modbusMaster.Quantity := addresses[i].length;
modbusMaster.MBAddr := addresses[i].start;
modbusMaster.pMemoryAddr := ADR(values[offset]);
modbusMaster.Execute := execute;
CASE addresses[i].accessFunction OF
ReadCoils:
	length := (addresses[i].length + 7) / 8;
	modbusMaster.ReadCoils(cbLength := length);
ReadInputStatus:
	length := (addresses[i].length + 7) / 8;
	modbusMaster.ReadInputStatus(cbLength := length);
ReadInputRegs:
	length := 2 * addresses[i].length;
	modbusMaster.ReadInputRegs(cbLength := length);
END_CASE
modbusMasterBusy := modbusMaster.BUSY;
modbusMasterError := modbusMaster.Error;
modbusMasterErrorId := modbusMaster.ErrorId;
modbusMasterBytesRead := modbusMaster.cbRead;

IF modbusMasterBusy THEN
	execute := FALSE;
END_IF
modbusMasterReadyTrigger(CLK := modbusMasterBusy);

IF initScan THEN
	initScan := FALSE;
ELSE
	IF modbusMasterReadyTrigger.Q THEN
		offset := offset + length;
		i := i + 1;
		IF i >= n THEN
			initScan := TRUE;
			setValues := TRUE;
		ELSE
			execute := TRUE;
		END_IF
	END_IF
END_IF

IF setValues THEN
	j := 0;
	Heizkreis1_PumpeEin := values[j].0;
	Heizkreis2_PumpeEin := values[j].1;
	Heizkreis1_MischerAuf := values[j].2;
	Heizkreis1_MischerZu := values[j].3;
	Heizkreis2_MischerAuf := values[j].4;
	Heizkreis2_MischerZu := values[j].5;
	j := j + 1;
	Heizkreis0_PumpeEin := values[j].0;
	j := j + 1;
	Stoerung := values[j].4;
	j := j + 1;
	Heizkreis3_PumpeEin := values[j].1;
	Heizkreis4_PumpeEin := values[j].2;
	Heizkreis3_MischerAuf := values[j].3;
	Heizkreis3_MischerZu := values[j].4;
	Heizkreis4_MischerAuf := values[j].5;
	Heizkreis4_MischerZu := values[j].6;
	j := j + 1;
	TuerOffen := values[j].0;
	STB := values[j].1;
	NotAus := values[j].2;
	j := j + 1; KesselTemperatur := INT_TO_REAL(values[j]) / 2;
	j := j + 1; AbgasTemperatur := INT_TO_REAL(values[j]);
	j := j + 1; BoardTemperatur := INT_TO_REAL(values[j]) / 2;
	j := j + 1; RestSauerstoff := INT_TO_REAL(values[j]) / 10;
	j := j + 1; AussenTemperatur := INT_TO_REAL(values[j]) / 2;
	j := j + 3; SaugzugDrehzahl := INT_TO_REAL(values[j]);
	j := j + 1; StbTemperatur := INT_TO_REAL(values[j]) / 2;
	j := j + 1; Fuehler2Temperatur := INT_TO_REAL(values[j]) / 2;
	j := j + 6; Saugzug := INT_TO_REAL(values[j]);
	j := j + 3; Kesselstellgroesse := INT_TO_REAL(values[j]);
	j := j + 3; Heizkreis1_VoraufIst := INT_TO_REAL(values[j]) / 2;
	j := j + 1; Heizkreis1_VoraufSoll := INT_TO_REAL(values[j]) / 2;
	j := j + 1; Heizkreis1_Party := values[j];
	j := j + 1; Heizkreis1_RaumTemperatur := INT_TO_REAL(values[j]) / 2;
	j := j + 1; Heizkreis2_VoraufIst := INT_TO_REAL(values[j]) / 2;
	j := j + 1; Heizkreis2_VoraufSoll := INT_TO_REAL(values[j]) / 2;
	j := j + 1; Heizkreis2_Party := values[j];
	j := j + 1; Heizkreis2_RaumTemperatur := INT_TO_REAL(values[j]) / 2;
	j := j + 1; Heizkreis3_VoraufIst := INT_TO_REAL(values[j]) / 2;
	j := j + 1; Heizkreis3_VoraufSoll := INT_TO_REAL(values[j]) / 2;
	j := j + 1; Heizkreis3_Party := values[j];
	j := j + 1; Heizkreis3_RaumTemperatur := INT_TO_REAL(values[j]) / 2;
	j := j + 1; Heizkreis4_VoraufIst := INT_TO_REAL(values[j]) / 2;
	j := j + 1; Heizkreis4_VoraufSoll := INT_TO_REAL(values[j]) / 2;
	j := j + 1; Heizkreis4_Party := values[j];
	j := j + 1; Heizkreis4_RaumTemperatur := INT_TO_REAL(values[j]) / 2;
	j := j + 1; Boiler1_TemperaturOben := INT_TO_REAL(values[j]) / 2;
	j := j + 1; Boiler1_TemperaturSolarreferenz := INT_TO_REAL(values[j]) / 2;
	j := j + 1; Board_TemperaturPelletmodul := INT_TO_REAL(values[j]) / 2;
	j := j + 1; Betriebsstunden := values[j];
	setValues := FALSE;
END_IF
END_FUNCTION_BLOCK

(* POU FBs/FB_ANALYSE_VOLTAGE, ST *)
FUNCTION_BLOCK FB_ANALYSE_VOLTAGE
VAR_INPUT
	uliStartTimeNextLatch: ARRAY [0..1] OF UDINT;
	bWcState: BOOL;
END_VAR
VAR_IN_OUT
	iVoltage : ARRAY [0..9] OF INT;
END_VAR
VAR
	iBufferV: ARRAY [0..209] OF INT;
	iBufferT: ARRAY [0..209] OF T_DCTIME;
	i: INT;
	dctActSample: T_DCTIME;
	multiplier: T_DCTIME;
	dctSampleDelay: T_DCTIME;
	fbGETCURTASKINDEX: GETCURTASKINDEX;
	tCylceTime: T_DCTIME;
	tSampleTime: T_DCTIME;
	dctElSampleDelta: T_DCTIME;
	n: INT;
	m: INT;
	dctZeroPoint: ARRAY [1..2] OF T_DCTIME;
	bZeroPoint: ARRAY [1..2] OF BOOL;
	ui64Sub: T_ULARGE_INTEGER;
	ui64a: T_ULARGE_INTEGER;
	ui64b: T_ULARGE_INTEGER;
	dctZeroPointDelta: T_DCTIME;
	dctNextSample: T_DCTIME;
	uliStartTimeNextLatchLastCycle: ARRAY [0..1] OF UDINT;
	iBufferZeroSumV: INT;
	dctSampleTimePerV: T_DCTIME;
	dctSampleTimeOffset: T_DCTIME;
	ui64Add: T_ULARGE_INTEGER;
	diResultAdd: DINT;
	diResultSub: DINT;
	ui64Add1: T_ULARGE_INTEGER;
	ui64Sub1: T_ULARGE_INTEGER;
	ui64Cmp1: T_ULARGE_INTEGER;
	iActVoltage: INT;
	tHalfCylceTime: T_DCTIME;
	multi: T_ULARGE_INTEGER;
END_VAR
VAR_OUTPUT
	lrFrequency: LREAL;
	tNextZeroVoltage: T_DCTIME;
	bError: BOOL;
	bZeroFound: BOOL;
	bZeroNow: BOOL;
END_VAR
VAR CONSTANT
	uiOversampling: UINT := 10;
END_VAR
MEMCPY(ADR(dctNextSample), ADR(uliStartTimeNextLatch), SIZEOF(dctActsample));
MEMCPY(ADR(ui64a), ADR(dctNextSample), SIZEOF(ui64a));
MEMCPY(ADR(ui64b), ADR(dctActSample), SIZEOF(ui64b));
ui64Sub := UInt64Sub64(ui64a, ui64b);
MEMCPY(ADR(dctElSampleDelta), ADR(ui64Sub), SIZEOF(dctElSampleDelta));

fbGETCURTASKINDEX(index => );
tCylceTime.dwLowPart := SYSTEMTASKINFOARR[fbGETCURTASKINDEX.index].cycleTime * 100;
tCylceTime.dwHighPart := 0;


IF (dctElSampleDelta.dwLowPart <> tCylceTime.dwLowPart)
OR (dctElSampleDelta.dwHighPart <> tCylceTime.dwHighPart) THEN
	bError := TRUE;
ELSE
	bError := FALSE;
END_IF

IF NOT bWcState AND NOT bError THEN
	(* Samplezeit *)
	IF uiOversampling > 0 THEN
		tSampleTime.dwLowPart := (SYSTEMTASKINFOARR[fbGETCURTASKINDEX.index].cycleTime*100)/uiOversampling;
		tSampleTime.dwHighPart := 0;
	END_IF

	(* Spannungsspeicher befüllen *)
	FOR i := 10 TO 209 DO
		iBufferV[i-10] := iBufferV[i];
		iBufferT[i-10] := iBufferT[i];
	END_FOR

	FOR i := 200 TO 209 DO
		multiplier := LREAL_TO_UINT64(INT_TO_LREAL(i-200));
		dctSampleDelay := UInt64Mul64(tSampleTime, multiplier);
		iBufferT[i] := UInt64Add64(dctActSample, dctSampleDelay);
		iBufferV[i] := iVoltage[i-200];
	END_FOR

	(* Zeit der Nulldurchgänge bestimmen *)
	m := 208;
	bZeroPoint[1] := FALSE;
	bZeroPoint[2] := FALSE;
	bZeroNow := FALSE;
	iActVoltage := iBufferV[200];
	FOR n := 1 TO 2 DO
		FOR i := m TO 0 BY -1 DO
			IF (iBufferV[i].15 AND NOT iBufferV[i+1].15) OR (NOT iBufferV[i].15 AND iBufferV[i+1].15) THEN
				iBufferZeroSumV := ABS(iBufferV[i]) + ABS(iBufferV[i+1]);
				IF iBufferZeroSumV > 0 THEN
					dctSampleTimePerV.dwLowPart := LREAL_TO_DWORD(DWORD_TO_LREAL(tSampleTime.dwLowPart) / INT_TO_LREAL(iBufferZeroSumV));
					dctSampleTimePerV.dwHighPart := 0;
					dctSampleTimeOffset := UInt64Mul64(dctSampleTimePerV, LREAL_TO_UINT64(INT_TO_LREAL(ABS(iBufferV[i]))));
					dctZeroPoint[n] := UInt64Add64(iBufferT[i], dctSampleTimeOffset);
				ELSE
					dctZeroPoint[n] := iBufferT[i];
				END_IF

				m := i-1;

				bZeroPoint[n] := TRUE;
				IF n = 1 THEN
					multi.dwLowPart := 1;
					tHalfCylceTime.dwLowPart := tCylceTime.dwLowPart/2;
					ui64Add1 := UInt64Add64(UInt64Add64(dctZeroPoint[n],UInt64Mul64(dctZeroPointDelta, multi)), tHalfCylceTime);
					ui64Sub1 := UInt64Sub64(UInt64Add64(dctZeroPoint[n],UInt64Mul64(dctZeroPointDelta, multi)), tHalfCylceTime);
					ui64Cmp1 := F_GetActualDcTime();
					diResultAdd := UInt64Cmp64(ui64Cmp1, ui64Add1);
					diResultSub := UInt64Cmp64(ui64Cmp1, ui64Sub1);
					IF (diResultSub >= 0) AND (diResultAdd <= 0)THEN
						bZeroNow := TRUE;
					END_IF
				END_IF
				EXIT;
			END_IF
		END_FOR
	END_FOR
	IF bZeroPoint[1] AND bZeroPoint[2] THEN

		(* Berechnung des nächsten Nullpunkts *)
		MEMCPY(ADR(ui64a), ADR(dctZeroPoint[1]), SIZEOF(ui64a));
		MEMCPY(ADR(ui64b), ADR(dctZeroPoint[2]), SIZEOF(ui64b));
		ui64Sub := UInt64Sub64(ui64a, ui64b);
		MEMCPY(ADR(dctZeroPointDelta), ADR(ui64Sub), SIZEOF(dctZeroPointDelta));

		MEMCPY(ADR(ui64a), ADR(dctZeroPointDelta), SIZEOF(ui64a));
		MEMCPY(ADR(ui64b), ADR(dctZeroPoint), SIZEOF(ui64b));
		ui64Add := UInt64Add64(ui64a, ui64b);
		MEMCPY(ADR(tNextZeroVoltage), ADR(ui64Add), SIZEOF(tNextZeroVoltage));


		lrFrequency := 1 / (2 * DWORD_TO_LREAL(dctZeroPointDelta.dwLowPart) / 1000000000);
	END_IF
END_IF
MEMCPY(ADR(dctActSample), ADR(uliStartTimeNextLatch), SIZEOF(dctActsample));

uliStartTimeNextLatchLastCycle := uliStartTimeNextLatch;
END_FUNCTION_BLOCK

(* POU FBs/FB_SYNC_RELAIS, ST *)
FUNCTION_BLOCK FB_SYNC_RELAIS
VAR_INPUT
	bValue: BOOL;
	udiDelayNanoSek: UDINT;
	tNextZeroVoltage: T_DCTIME;
END_VAR
VAR_OUTPUT
	bRelay AT %Q*: BOOL;
END_VAR
VAR
	fbGETCURTASKINDEX: GETCURTASKINDEX;
	tNextZeroVoltageLast: T_DCTIME;
	TON_FAILURE: TON;
	TOF_WAIT: TOF;
	udiLastOnlineChangeCount: UDINT;
	multi: T_DCTIME;
	ui64Add1: T_ULARGE_INTEGER;
	tHalfCylceTime: T_DCTIME;
	ui64Sub1: T_ULARGE_INTEGER;
	ui64Cmp1: T_ULARGE_INTEGER;
	diResultAdd: DINT;
	diResultSub: DINT;
	tCylceTime: T_DCTIME;
END_VAR
(*fTvalue(CLK:=bValue AND bRelay);
IF fTvalue.Q OR bReset THEN
	bRelay := FALSE;
	bReset := FALSE;
END_IF
*)

TON_FAILURE(IN := tNextZeroVoltage.dwLowPart = tNextZeroVoltageLast.dwLowPart, PT := t#100ms);
tNextZeroVoltageLast.dwLowPart := tNextZeroVoltage.dwLowPart;

TOF_WAIT(IN := SYSTEMINFO.onlineChangeCount <> udiLastOnlineChangeCount, PT := t#0.5s);
udiLastOnlineChangeCount := SYSTEMINFO.onlineChangeCount;

IF bValue AND NOT bRelay AND NOT TON_FAILURE.Q THEN
	fbGETCURTASKINDEX(index => );
	tCylceTime.dwLowPart := SYSTEMTASKINFOARR[fbGETCURTASKINDEX.index].cycleTime * 100;
	tCylceTime.dwHighPart := 0;

	multi.dwLowPart := udiDelayNanoSek;
	tHalfCylceTime.dwLowPart := tCylceTime.dwLowPart/2;
	ui64Add1 := UInt64Add64(UInt64Sub64(tNextZeroVoltage, multi), tHalfCylceTime);
	ui64Sub1 := UInt64Sub64(UInt64Sub64(tNextZeroVoltage, multi), tHalfCylceTime);
	ui64Cmp1 := F_GetActualDcTime();
	diResultAdd := UInt64Cmp64(ui64Cmp1, ui64Add1);
	diResultSub := UInt64Cmp64(ui64Cmp1, ui64Sub1);

	IF (diResultSub >= 0) AND (diResultAdd <= 0) THEN
		bRelay := TRUE;
	END_IF
END_IF

IF NOT bValue AND bRelay AND NOT TON_FAILURE.Q THEN
	fbGETCURTASKINDEX(index => );
	tCylceTime.dwLowPart := SYSTEMTASKINFOARR[fbGETCURTASKINDEX.index].cycleTime * 100;
	tCylceTime.dwHighPart := 0;

	multi.dwLowPart := udiDelayNanoSek / 2;
	tHalfCylceTime.dwLowPart := tCylceTime.dwLowPart / 2;
	ui64Add1 := UInt64Add64(UInt64Sub64(tNextZeroVoltage, multi), tHalfCylceTime);
	ui64Sub1 := UInt64Sub64(UInt64Sub64(tNextZeroVoltage, multi), tHalfCylceTime);
	ui64Cmp1 := F_GetActualDcTime();
	diResultAdd := UInt64Cmp64(ui64Cmp1, ui64Add1);
	diResultSub := UInt64Cmp64(ui64Cmp1, ui64Sub1);

	IF (diResultSub >= 0) AND (diResultAdd <= 0)THEN
		bRelay := FALSE;
	END_IF
END_IF
END_FUNCTION_BLOCK

(* POU FBs/FB_Modbus_RTU_Master_KL6x22B, ST *)
FUNCTION_BLOCK FB_Modbus_RTU_Master_KL6x22B
VAR_INPUT
	bStart: BOOL; (* Start Modbus-Communication *)
	byModbusSlaveStartAdress: BYTE := 1; (* First Modbus Device Address *)
	byModbusSlaveEndAdress: BYTE := 247; (* Last Modbus Device Address *)
	tModbusSlaveTimeout: TIME := t#500ms; (* Modbus Communication Timeout *)
	tDelayModbusTime: TIME := t#50ms; (* Delay between two Modbus Requests *)
	bIgnoreError: BOOL; (* Ignore ever Modbus Error *)
END_VAR
VAR_OUTPUT
	bBusy: BOOL; (* if TRUE, Modbustelegramms are being sent *)
	bError: BOOL; (* if TRUE, a Modbustelegramm wasn't send correctly *)
	eErrorID: MODBUS_ERRORS;
	bNoResponse: BOOL; (* if TRUE, a FB with a DeviceAddress isn't existing as phyical device *)
	byLastNoResponseModbusAddress: BYTE;
END_VAR
VAR_IN_OUT
	stCommunication: stFB_ModbusMaster; (* Communicationvariable must connect with ever Slave FB *)
END_VAR
VAR
	FB_ModbusRtuMaster_KL6x22B: ModbusRtuMaster_KL6x22B;
	R_TRIG_START: R_TRIG;
	F_TRIG_ModbusReady: F_TRIG;
	TON_Delay: TON;
	i: INT;
	j: INT;
	bBusyMaster: BOOL;
	bNextModbusDevice: BOOL;
	bNextData: BOOL;
END_VAR
R_TRIG_START(CLK := bStart);
TON_Delay(IN := i = 2, PT := tDelayModbusTime);

F_TRIG_ModbusReady(CLK := FB_ModbusRtuMaster_KL6x22B.BUSY);
IF F_TRIG_ModbusReady.Q THEN
	bBusy := FALSE;
END_IF

(* Init FB *)
IF R_TRIG_START.Q THEN
	i := 0;
END_IF

CASE i OF
0: (* Set Startaddress *)
	IF R_TRIG_START.Q THEN
		bBusy := TRUE;
		bError := FALSE;
		eErrorID := 0;
		stCommunication.byCurrentModbusSlaveAdress := byModbusSlaveStartAdress;
		i := i + 1;
	END_IF
1: (* Exist Address?*)
	IF stCommunication.bModbusAddressExist THEN
		i := i + 1;
		stCommunication.bModbusCommunicationActive := TRUE;
	ELSE
		j := j + 1;
	END_IF
	IF j > 10 THEN
		stCommunication.byCurrentModbusSlaveAdress := stCommunication.byCurrentModbusSlaveAdress + 1;
		j := 0;
	END_IF
	IF stCommunication.byCurrentModbusSlaveAdress > byModbusSlaveEndAdress OR stCommunication.byCurrentModbusSlaveAdress > 247 THEN
		stCommunication.byCurrentModbusSlaveAdress := byModbusSlaveStartAdress;
		IF byModbusSlaveStartAdress < 1 THEN
			stCommunication.byCurrentModbusSlaveAdress := 1;
		END_IF
	END_IF

2: (* Init Modbus and order data from slave*)
	IF TON_Delay.Q AND bStart THEN
		bBusy := TRUE;
		bError := FALSE;
		eErrorID := 0;
		FB_ModbusRtuMaster_KL6x22B.ReadCoils(Execute := FALSE);
		FB_ModbusRtuMaster_KL6x22B.ReadInputStatus(Execute := FALSE);
		FB_ModbusRtuMaster_KL6x22B.ReadRegs(Execute := FALSE);
		FB_ModbusRtuMaster_KL6x22B.ReadInputRegs(Execute := FALSE);
		FB_ModbusRtuMaster_KL6x22B.WriteSingleCoil(Execute := FALSE);
		FB_ModbusRtuMaster_KL6x22B.WriteSingleRegister(Execute := FALSE);
		FB_ModbusRtuMaster_KL6x22B.Diagnostics(Execute := FALSE);
		FB_ModbusRtuMaster_KL6x22B.WriteMultipleCoils(Execute := FALSE);
		FB_ModbusRtuMaster_KL6x22B.WriteRegs(Execute := FALSE);
		i := i + 1;
	END_IF
3: (*Wait for new data from slave *)
	CASE stCommunication.stCurrentDeviceSpace[0].iModbusFunction OF
		1:
			FB_ModbusRtuMaster_KL6x22B.ReadCoils(
				UnitID:=stCommunication.byCurrentModbusSlaveAdress,
				Quantity:= stCommunication.stCurrentDeviceSpace[0].wSPSDataSpaceLength/2,
				MBAddr:= stCommunication.stCurrentDeviceSpace[0].wModbusAdress,
				cbLength:= stCommunication.stCurrentDeviceSpace[0].wSPSDataSpaceLength,
				pMemoryAddr:= stCommunication.stCurrentDeviceSpace[0].pSPSDataSpace,
				Execute:= TRUE,
				Timeout := tModbusSlaveTimeout,
				Busy=>bBusyMaster);
		2:
			FB_ModbusRtuMaster_KL6x22B.ReadInputStatus(
				UnitID:=stCommunication.byCurrentModbusSlaveAdress,
				Quantity:= stCommunication.stCurrentDeviceSpace[0].wSPSDataSpaceLength/2,
				MBAddr:= stCommunication.stCurrentDeviceSpace[0].wModbusAdress,
				cbLength:= stCommunication.stCurrentDeviceSpace[0].wSPSDataSpaceLength,
				pMemoryAddr:= stCommunication.stCurrentDeviceSpace[0].pSPSDataSpace,
				Execute:= TRUE,
				Timeout := tModbusSlaveTimeout,
				Busy=>bBusyMaster);
		3:
			FB_ModbusRtuMaster_KL6x22B.ReadRegs(
				UnitID:=stCommunication.byCurrentModbusSlaveAdress,
				Quantity:= stCommunication.stCurrentDeviceSpace[0].wSPSDataSpaceLength/2,
				MBAddr:= stCommunication.stCurrentDeviceSpace[0].wModbusAdress,
				cbLength:= stCommunication.stCurrentDeviceSpace[0].wSPSDataSpaceLength,
				pMemoryAddr:= stCommunication.stCurrentDeviceSpace[0].pSPSDataSpace,
				Execute:= TRUE,
				Timeout := tModbusSlaveTimeout,
				Busy=>bBusyMaster);
		4:
			FB_ModbusRtuMaster_KL6x22B.ReadInputRegs(
				UnitID:=stCommunication.byCurrentModbusSlaveAdress,
				Quantity:= stCommunication.stCurrentDeviceSpace[0].wSPSDataSpaceLength/2,
				MBAddr:= stCommunication.stCurrentDeviceSpace[0].wModbusAdress,
				cbLength:= stCommunication.stCurrentDeviceSpace[0].wSPSDataSpaceLength,
				pMemoryAddr:= stCommunication.stCurrentDeviceSpace[0].pSPSDataSpace,
				Execute:= TRUE,
				Timeout := tModbusSlaveTimeout,
				Busy=>bBusyMaster);
		5:
			FB_ModbusRtuMaster_KL6x22B.WriteSingleCoil(
				UnitID:=stCommunication.byCurrentModbusSlaveAdress,
				Quantity:= stCommunication.stCurrentDeviceSpace[0].wSPSDataSpaceLength/2,
				MBAddr:= stCommunication.stCurrentDeviceSpace[0].wModbusAdress,
				cbLength:= stCommunication.stCurrentDeviceSpace[0].wSPSDataSpaceLength,
				pMemoryAddr:= stCommunication.stCurrentDeviceSpace[0].pSPSDataSpace,
				Execute:= TRUE,
				Timeout := tModbusSlaveTimeout,
				Busy=>bBusyMaster);
		6:
			FB_ModbusRtuMaster_KL6x22B.WriteSingleRegister(
				UnitID:=stCommunication.byCurrentModbusSlaveAdress,
				Quantity:= stCommunication.stCurrentDeviceSpace[0].wSPSDataSpaceLength/2,
				MBAddr:= stCommunication.stCurrentDeviceSpace[0].wModbusAdress,
				cbLength:= stCommunication.stCurrentDeviceSpace[0].wSPSDataSpaceLength,
				pMemoryAddr:= stCommunication.stCurrentDeviceSpace[0].pSPSDataSpace,
				Execute:= TRUE,
				Timeout := tModbusSlaveTimeout,
				Busy=>bBusyMaster);
		8:
			FB_ModbusRtuMaster_KL6x22B.Diagnostics(
				UnitID:=stCommunication.byCurrentModbusSlaveAdress,
				Quantity:= stCommunication.stCurrentDeviceSpace[0].wSPSDataSpaceLength/2,
				MBAddr:= stCommunication.stCurrentDeviceSpace[0].wModbusAdress,
				cbLength:= stCommunication.stCurrentDeviceSpace[0].wSPSDataSpaceLength,
				pMemoryAddr:= stCommunication.stCurrentDeviceSpace[0].pSPSDataSpace,
				Execute:= TRUE,
				Timeout := tModbusSlaveTimeout,
				Busy=>bBusyMaster);
		15:
			FB_ModbusRtuMaster_KL6x22B.WriteMultipleCoils(
				UnitID:=stCommunication.byCurrentModbusSlaveAdress,
				Quantity:= stCommunication.stCurrentDeviceSpace[0].wSPSDataSpaceLength/2,
				MBAddr:= stCommunication.stCurrentDeviceSpace[0].wModbusAdress,
				cbLength:= stCommunication.stCurrentDeviceSpace[0].wSPSDataSpaceLength,
				pMemoryAddr:= stCommunication.stCurrentDeviceSpace[0].pSPSDataSpace,
				Execute:= TRUE,
				Timeout := tModbusSlaveTimeout,
				Busy=>bBusyMaster);
		16:
			FB_ModbusRtuMaster_KL6x22B.WriteRegs(
				UnitID:=stCommunication.byCurrentModbusSlaveAdress,
				Quantity:= stCommunication.stCurrentDeviceSpace[0].wSPSDataSpaceLength/2,
				MBAddr:= stCommunication.stCurrentDeviceSpace[0].wModbusAdress,
				cbLength:= stCommunication.stCurrentDeviceSpace[0].wSPSDataSpaceLength,
				pMemoryAddr:= stCommunication.stCurrentDeviceSpace[0].pSPSDataSpace,
				Execute:= TRUE,
				Timeout := tModbusSlaveTimeout,
				Busy=>bBusyMaster);
	ELSE
		bError := TRUE;
		eErrorID := 1;
	END_CASE

	IF F_TRIG_ModbusReady.Q AND NOT FB_ModbusRtuMaster_KL6x22B.Error THEN (*No Error*)
		bNoResponse := FALSE;
		bError := FALSE;
		bNextData := TRUE;
	ELSIF FB_ModbusRtuMaster_KL6x22B.Error AND FB_ModbusRtuMaster_KL6x22B.ErrorId = 16#25 THEN (*no  Response *)
		i := 1;
		bNoResponse := TRUE;
		bError := TRUE;
		eErrorID := FB_ModbusRtuMaster_KL6x22B.ErrorId;
		byLastNoResponseModbusAddress := stCommunication.byCurrentModbusSlaveAdress;
		stCommunication.byCurrentModbusSlaveAdress := stCommunication.byCurrentModbusSlaveAdress + 1;
		stCommunication.bModbusAddressExist := FALSE;
		stCommunication.bModbusCommunicationActive := FALSE;
		i := 1;
		FOR j := 0 TO stCommunication.iNumberOfData DO
			stCommunication.stCurrentDeviceSpace[stCommunication.iNumberOfData].iModbusFunction := 0;
			stCommunication.stCurrentDeviceSpace[stCommunication.iNumberOfData].pSPSDataSpace := 0;
			stCommunication.stCurrentDeviceSpace[stCommunication.iNumberOfData].wModbusAdress := 0;
			stCommunication.stCurrentDeviceSpace[stCommunication.iNumberOfData].wSPSDataSpaceLength := 0;
		END_FOR
	ELSIF FB_ModbusRtuMaster_KL6x22B.Error AND bIgnoreError THEN
		bNoResponse := FALSE;
		bError := TRUE;
		bNextData := TRUE;
	ELSIF FB_ModbusRtuMaster_KL6x22B.Error THEN
		i := 100;
	END_IF

	IF bNextData THEN
		FOR j := 1 TO stCommunication.iNumberOfData DO
			stCommunication.stCurrentDeviceSpace[j-1] := stCommunication.stCurrentDeviceSpace[j];
		END_FOR
		stCommunication.stCurrentDeviceSpace[stCommunication.iNumberOfData].iModbusFunction := 0;
		stCommunication.stCurrentDeviceSpace[stCommunication.iNumberOfData].pSPSDataSpace := 0;
		stCommunication.stCurrentDeviceSpace[stCommunication.iNumberOfData].wModbusAdress := 0;
		stCommunication.stCurrentDeviceSpace[stCommunication.iNumberOfData].wSPSDataSpaceLength := 0;
		i := 2;
		bNextData := FALSE;
		bBusy := FALSE;
		IF stCommunication.stCurrentDeviceSpace[0].iModbusFunction = 0 THEN
			stCommunication.byCurrentModbusSlaveAdress := stCommunication.byCurrentModbusSlaveAdress + 1;
			stCommunication.bModbusAddressExist := FALSE;
			stCommunication.bModbusCommunicationActive := FALSE;
			i := 1;
		END_IF
	END_IF
100:
	bError := FB_ModbusRtuMaster_KL6x22B.Error;
	eErrorID := FB_ModbusRtuMaster_KL6x22B.ErrorId;
END_CASE
END_FUNCTION_BLOCK

(* POU FBs/FB_ScanModbusSlaveAdresses_KL6x22B, ST *)
FUNCTION_BLOCK FB_ScanModbusSlaveAdresses_KL6x22B
VAR_INPUT
	bStartScan: BOOL; (* Start scanning *)
	bOnlyRead: BOOL;
	byModbusSlaveDeviceAdress: BYTE := 1; (* Modbus Device Address *)
	MBStartAddr: WORD := 0; (* First ModbusRegisterAddress *)
	MBEndAddr: WORD := 100; (* Last ModbusRegisterAddress *)
	(* ATTENTION please!!! This FB writes to the ModbusRegisterAddress
		the value 0 with every write function!!!
		DON'T SCAN SYSTEMREGISTER OR FIRMWARE REGISTER
		... the Device could be destroyed! *)
END_VAR
VAR_OUTPUT
	rPercentOfScanProzess: REAL;
	bNoFreeSpaceForNewValues: BOOL;
	bReady: BOOL;
	stValues: ARRAY [0..999] OF stResultOfModbusSlaveScan; (* Scanresult *)
END_VAR
VAR
	FB_ModbusRtuMaster_KL6x22B: ModbusRtuMaster_KL6x22B;
	F_TRIG1: F_TRIG;
	R_TRIG1: R_TRIG;
	F_TRIG2: F_TRIG;
	bStart: BOOL;
	MBFunction: INT := 1;
	MBAddr: WORD;
	Pos: INT;
	i: INT;
	Result: UDINT;
	rActuellScanProzess: REAL;
END_VAR
CASE MBFunction OF
1:
	FB_ModbusRtuMaster_KL6x22B.ReadCoils(
		UnitID := byModbusSlaveDeviceAdress,
		Quantity := 1,
		MBAddr := MBAddr,
		cbLength := 2,
		pMemoryAddr := ADR(stValues[Pos].wValue),
		Execute := bStart,
		Timeout := t#1s,
		BUSY => ,
		Error => ,
		ErrorId => ,
		cbRead => );
2:
	FB_ModbusRtuMaster_KL6x22B.ReadInputStatus(
		UnitID:=byModbusSlaveDeviceAdress ,
		Quantity:=1 ,
		MBAddr:=MBAddr ,
		cbLength:=2 ,
		pMemoryAddr:=ADR(stValues[Pos].wValue) ,
		Execute:=bStart ,
		Timeout:=t#1s ,
		BUSY=> ,
		Error=> ,
		ErrorId=> ,
		cbRead=> );
3:
	FB_ModbusRtuMaster_KL6x22B.ReadRegs(
		UnitID:=byModbusSlaveDeviceAdress ,
		Quantity:=1 ,
		MBAddr:=MBAddr ,
		cbLength:=2 ,
		pMemoryAddr:=ADR(stValues[Pos].wValue) ,
		Execute:=bStart ,
		Timeout:=t#1s ,
		BUSY=> ,
		Error=> ,
		ErrorId=> ,
		cbRead=> );
4:
	FB_ModbusRtuMaster_KL6x22B.ReadInputRegs(
		UnitID:=byModbusSlaveDeviceAdress ,
		Quantity:=1 ,
		MBAddr:=MBAddr ,
		cbLength:=2 ,
		pMemoryAddr:=ADR(stValues[Pos].wValue) ,
		Execute:=bStart ,
		Timeout:=t#1s ,
		BUSY=> ,
		Error=> ,
		ErrorId=> ,
		cbRead=> );
5:
	FB_ModbusRtuMaster_KL6x22B.WriteSingleCoil(
		UnitID:=byModbusSlaveDeviceAdress ,
		Quantity:=1 ,
		MBAddr:=MBAddr ,
		cbLength:=2 ,
		pMemoryAddr:=ADR(stValues[Pos].wValue) ,
		Execute:=bStart ,
		Timeout:=t#1s ,
		BUSY=> ,
		Error=> ,
		ErrorId=> ,
		cbRead=> );
6:
	FB_ModbusRtuMaster_KL6x22B.WriteSingleRegister(
		UnitID:=byModbusSlaveDeviceAdress ,
		Quantity:=1 ,
		MBAddr:=MBAddr ,
		cbLength:=2 ,
		pMemoryAddr:=ADR(stValues[Pos].wValue) ,
		Execute:=bStart ,
		Timeout:=t#1s ,
		BUSY=> ,
		Error=> ,
		ErrorId=> ,
		cbRead=> );
8:
	FB_ModbusRtuMaster_KL6x22B.Diagnostics(
		UnitID:=byModbusSlaveDeviceAdress ,
		Quantity:=1 ,
		MBAddr:=MBAddr ,
		cbLength:=2 ,
		pMemoryAddr:=ADR(stValues[Pos].wValue) ,
		Execute:=bStart ,
		Timeout:=t#1s ,
		BUSY=> ,
		Error=> ,
		ErrorId=> ,
		cbRead=> );
15:
	FB_ModbusRtuMaster_KL6x22B.WriteMultipleCoils(
		UnitID:=byModbusSlaveDeviceAdress ,
		Quantity:=1 ,
		MBAddr:=MBAddr ,
		cbLength:=2 ,
		pMemoryAddr:=ADR(stValues[Pos].wValue) ,
		Execute:=bStart ,
		Timeout:=t#1s ,
		BUSY=> ,
		Error=> ,
		ErrorId=> ,
		cbRead=> );
16:
	FB_ModbusRtuMaster_KL6x22B.WriteRegs(
		UnitID:=byModbusSlaveDeviceAdress ,
		Quantity:=1 ,
		MBAddr:=MBAddr ,
		cbLength:=2 ,
		pMemoryAddr:=ADR(stValues[Pos].wValue) ,
		Execute:=bStart ,
		Timeout:=t#1s ,
		BUSY=> ,
		Error=> ,
		ErrorId=> ,
		cbRead=> );
END_CASE

F_TRIG1(CLK := FB_ModbusRtuMaster_KL6x22B.BUSY);

R_TRIG1(CLK := bStartScan);
F_TRIG2(CLK := bStartScan);

IF F_TRIG2.Q THEN
	i := 0;
END_IF

CASE i OF
0:
	IF R_TRIG1.Q THEN
		i := i + 1;
		bStart := FALSE;
		bNoFreeSpaceForNewValues := FALSE;
		bReady := FALSE;
		MBAddr := MBStartAddr;
		rPercentOfScanProzess := 0.0;
		rActuellScanProzess := 0.0;
	END_IF
1:
	bStart := TRUE;
	i := i + 1;
2:
	IF F_TRIG1.Q AND ((NOT FB_ModbusRtuMaster_KL6x22B.Error) OR FB_ModbusRtuMaster_KL6x22B.ErrorId = 3) THEN
		stValues[Pos].eModbusError := FB_ModbusRtuMaster_KL6x22B.ErrorId;
		stValues[Pos].eModbusfunction := MBFunction;
		stValues[Pos].iModbusAdress := MBAddr;
		(*New Array Position*)
		Pos := Pos + 1;
	END_IF

	IF F_TRIG1.Q THEN
		IF Pos > 999 THEN
			Pos := 0;
			i := 0;
			bNoFreeSpaceForNewValues := TRUE;
		END_IF

		MBAddr := MBAddr + 1;
		i := 1;
		bStart := FALSE;
		IF MBAddr > MBEndAddr THEN
			MBAddr := MBStartAddr;
			MBFunction := MBFunction + 1;
			IF MBFunction > 4 AND bOnlyRead OR MBFunction = 17 THEN
				MBFunction := 1;
				i := 4;
				bReady := TRUE;
			ELSE
				IF MBFunction = 7 THEN
					MBFunction := 8;
				ELSIF MBFunction = 9 THEN
					MBFunction := 15;
				ELSE
					;
				END_IF
			END_IF
		END_IF
	END_IF
4:
		rPercentOfScanProzess := 100.0;
END_CASE

IF F_TRIG1.Q THEN
	rActuellScanProzess := rActuellScanProzess + 1.0;
END_IF

IF NOT (i = 4) THEN
	rPercentOfScanProzess := (100.0 * rActuellScanProzess) / (9.0 * WORD_TO_REAL(MBEndAddr - MBStartAddr));
END_IF
END_FUNCTION_BLOCK

(* POU FBs/FB_Toggle, ST *)
FUNCTION_BLOCK FB_Toggle
VAR_INPUT
	onTime: TIME :=  t#0.5s;
	offTime: TIME := t#1s;
END_VAR
VAR_OUTPUT
	Q: BOOL;
END_VAR
VAR
	t1: TON;
	t2: TOF;
END_VAR
t1(IN := NOT t2.Q, pt := offTime);
t2(IN := t1.Q, pt := onTime);
Q := t2.Q;

(* c.henke variant:
TON1(IN := NOT TON1.Q AND bStart, PT := t#1s);
IF TON1.Q THEN
	bRelayPLC := NOT bRelayPLC;
END_IF
*)
END_FUNCTION_BLOCK

(* Visualisation VI_BACKGROUND
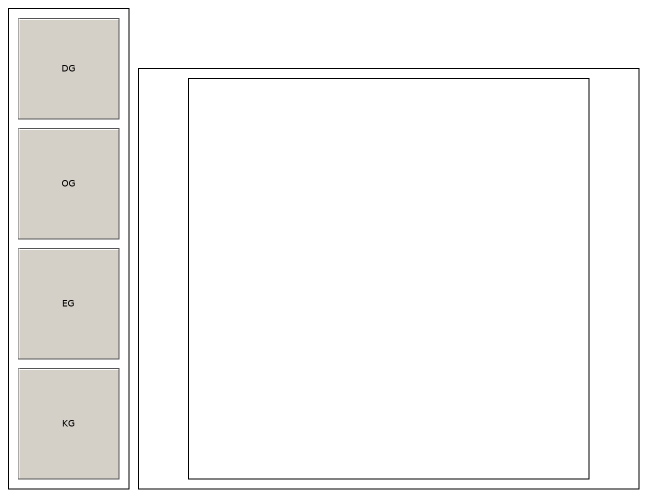
button at (10,360)-(111,471): text "KG"; opens vi_KG
button at (10,240)-(111,351): text "EG"; opens vi_EG
button at (10,120)-(111,231): text "OG"; opens vi_OG
button at (10,10)-(111,111): text "DG"; opens vi_DG
3 more shapes without text or variables
*)

(* Visualisation templates/VI_BUTTONDOUBLE
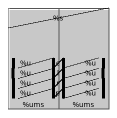
button at (50,0)-(101,101): text "%ums"; shows $fbButton_R$.LONGPRESS; taps $fbButton_R$.viIN
button at (0,0)-(51,101): text "%ums"; shows $fbButton_L$.LONGPRESS; taps $fbButton_L$.viIN
curve at (55,80)-(90,90): text "%u"; shows $fbButton_R$.usageCounterPress
curve at (95,80)-(95,90): alarm colour if $fbButton_R$.toggleOnPress
curve at (95,70)-(95,80): alarm colour if $fbButton_R$.toggleOnRelease
curve at (95,60)-(95,70): alarm colour if $fbButton_R$.toggleOnLongpress
curve at (95,50)-(95,60): alarm colour if $fbButton_R$.toggleOnClick
curve at (55,70)-(90,80): text "%u"; shows $fbButton_R$.usageCounterRelease
curve at (55,60)-(90,70): text "%u"; shows $fbButton_R$.usageCounterLongpress
curve at (55,50)-(90,60): text "%u"; shows $fbButton_R$.usageCounterClick
curve at (55,80)-(55,90): alarm colour if $fbButton_R$.isPressed
curve at (55,70)-(55,80): alarm colour if $fbButton_R$.isReleased
curve at (55,60)-(55,70): alarm colour if $fbButton_R$.isLongpressed
curve at (55,50)-(55,60): alarm colour if $fbButton_R$.isClicked
curve at (45,50)-(55,60): text "c"
curve at (45,60)-(55,70): text "l"
curve at (45,70)-(55,80): text "r"
curve at (45,80)-(55,90): text "p"
curve at (10,80)-(45,90): text "%u"; shows $fbButton_L$.usageCounterPress
curve at (5,80)-(5,90): alarm colour if $fbButton_L$.toggleOnPress
curve at (5,70)-(5,80): alarm colour if $fbButton_L$.toggleOnRelease
curve at (5,60)-(5,70): alarm colour if $fbButton_L$.toggleOnLongpress
curve at (5,50)-(5,60): alarm colour if $fbButton_L$.toggleOnClick
curve at (10,70)-(45,80): text "%u"; shows $fbButton_L$.usageCounterRelease
curve at (10,60)-(45,70): text "%u"; shows $fbButton_L$.usageCounterLongpress
curve at (10,50)-(45,60): text "%u"; shows $fbButton_L$.usageCounterClick
curve at (45,80)-(45,90): alarm colour if $fbButton_L$.isPressed
curve at (45,70)-(45,80): alarm colour if $fbButton_L$.isReleased
curve at (45,60)-(45,70): alarm colour if $fbButton_L$.isLongpressed
curve at (45,50)-(45,60): alarm colour if $fbButton_L$.isClicked
curve at (0,0)-(100,20): text "%s"; shows $fbButton_L$.viText
*)

(* Visualisation templates/vi_ButtonDouble_tiny
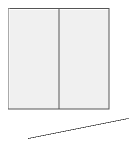
button at (50,0)-(101,101): taps $fbButton_R$.viIN
button at (0,0)-(51,101): taps $fbButton_L$.viIN
1 more shapes without text or variables
*)

(* Visualisation templates/vi_ButtonSingle
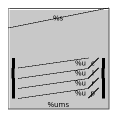
button at (0,0)-(101,101): text "%ums"; shows $fbButton$.LONGPRESS; taps $fbButton$.viIN
curve at (0,0)-(100,20): text "%s"; shows $fbButton$.viText
curve at (10,80)-(80,90): text "%u"; shows $fbButton$.usageCounterPress
curve at (95,80)-(95,90): alarm colour if $fbButton$.toggleOnPress
curve at (95,70)-(95,80): alarm colour if $fbButton$.toggleOnRelease
curve at (95,60)-(95,70): alarm colour if $fbButton$.toggleOnLongpress
curve at (95,50)-(95,60): alarm colour if $fbButton$.toggleOnClick
curve at (10,70)-(80,80): text "%u"; shows $fbButton$.usageCounterRelease
curve at (10,60)-(80,70): text "%u"; shows $fbButton$.usageCounterLongpress
curve at (10,50)-(80,60): text "%u"; shows $fbButton$.usageCounterClick
curve at (80,50)-(90,60): text "c"
curve at (80,60)-(90,70): text "l"
curve at (80,70)-(90,80): text "r"
curve at (80,80)-(90,90): text "p"
curve at (5,80)-(5,90): alarm colour if $fbButton$.isPressed
curve at (5,70)-(5,80): alarm colour if $fbButton$.isReleased
curve at (5,60)-(5,70): alarm colour if $fbButton$.isLongpressed
curve at (5,50)-(5,60): alarm colour if $fbButton$.isClicked
*)

(* Visualisation templates/vi_ButtonSingle_tiny
button at (0,0)-(101,101): taps $fbButton$.viIN
*)

(* Visualisation templates/vi_ButtonTripple
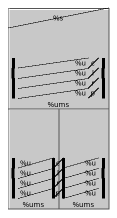
button at (50,100)-(101,201): text "%ums"; shows $fbButton_R$.LONGPRESS; taps $fbButton_R$.viIN
button at (0,100)-(51,201): text "%ums"; shows $fbButton_L$.LONGPRESS; taps $fbButton_L$.viIN
curve at (55,180)-(90,190): text "%u"; shows $fbButton_R$.usageCounterPress
curve at (95,180)-(95,190): alarm colour if $fbButton_R$.toggleOnPress
curve at (95,170)-(95,180): alarm colour if $fbButton_R$.toggleOnRelease
curve at (95,160)-(95,170): alarm colour if $fbButton_R$.toggleOnLongpress
curve at (95,150)-(95,160): alarm colour if $fbButton_R$.toggleOnClick
curve at (55,170)-(90,180): text "%u"; shows $fbButton_R$.usageCounterRelease
curve at (55,160)-(90,170): text "%u"; shows $fbButton_R$.usageCounterLongpress
curve at (55,150)-(90,160): text "%u"; shows $fbButton_R$.usageCounterClick
curve at (55,180)-(55,190): alarm colour if $fbButton_R$.isPressed
curve at (55,170)-(55,180): alarm colour if $fbButton_R$.isReleased
curve at (55,160)-(55,170): alarm colour if $fbButton_R$.isLongpressed
curve at (55,150)-(55,160): alarm colour if $fbButton_R$.isClicked
curve at (45,150)-(55,160): text "c"
curve at (45,160)-(55,170): text "l"
curve at (45,170)-(55,180): text "r"
curve at (45,180)-(55,190): text "p"
curve at (10,180)-(45,190): text "%u"; shows $fbButton_L$.usageCounterPress
curve at (5,180)-(5,190): alarm colour if $fbButton_L$.toggleOnPress
curve at (5,170)-(5,180): alarm colour if $fbButton_L$.toggleOnRelease
curve at (5,160)-(5,170): alarm colour if $fbButton_L$.toggleOnLongpress
curve at (5,150)-(5,160): alarm colour if $fbButton_L$.toggleOnClick
curve at (10,170)-(45,180): text "%u"; shows $fbButton_L$.usageCounterRelease
curve at (10,160)-(45,170): text "%u"; shows $fbButton_L$.usageCounterLongpress
curve at (10,150)-(45,160): text "%u"; shows $fbButton_L$.usageCounterClick
curve at (45,180)-(45,190): alarm colour if $fbButton_L$.isPressed
curve at (45,170)-(45,180): alarm colour if $fbButton_L$.isReleased
curve at (45,160)-(45,170): alarm colour if $fbButton_L$.isLongpressed
curve at (45,150)-(45,160): alarm colour if $fbButton_L$.isClicked
button at (0,0)-(101,101): text "%ums"; shows $fbButton_T$.LONGPRESS; taps $fbButton_T$.viIN
curve at (0,0)-(100,20): text "%s"; shows $fbButton_T$.viText
curve at (10,80)-(80,90): text "%u"; shows $fbButton_T$.usageCounterPress
curve at (95,80)-(95,90): alarm colour if $fbButton_T$.toggleOnPress
curve at (95,70)-(95,80): alarm colour if $fbButton_T$.toggleOnRelease
curve at (95,60)-(95,70): alarm colour if $fbButton_T$.toggleOnLongpress
curve at (95,50)-(95,60): alarm colour if $fbButton_T$.toggleOnClick
curve at (10,70)-(80,80): text "%u"; shows $fbButton_T$.usageCounterRelease
curve at (10,60)-(80,70): text "%u"; shows $fbButton_T$.usageCounterLongpress
curve at (10,50)-(80,60): text "%u"; shows $fbButton_T$.usageCounterClick
curve at (80,50)-(90,60): text "c"
curve at (80,60)-(90,70): text "l"
curve at (80,70)-(90,80): text "r"
curve at (80,80)-(90,90): text "p"
curve at (5,80)-(5,90): alarm colour if $fbButton_T$.isPressed
curve at (5,70)-(5,80): alarm colour if $fbButton_T$.isReleased
curve at (5,60)-(5,70): alarm colour if $fbButton_T$.isLongpressed
curve at (5,50)-(5,60): alarm colour if $fbButton_T$.isClicked
*)

(* Visualisation templates/vi_ButtonTripple_tiny
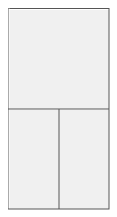
button at (50,100)-(101,201): taps $fbButton_R$.viIN
button at (0,100)-(51,201): taps $fbButton_L$.viIN
button at (0,0)-(101,101): taps $fbButton_T$.viIN
*)

(* Visualisation VI_DG
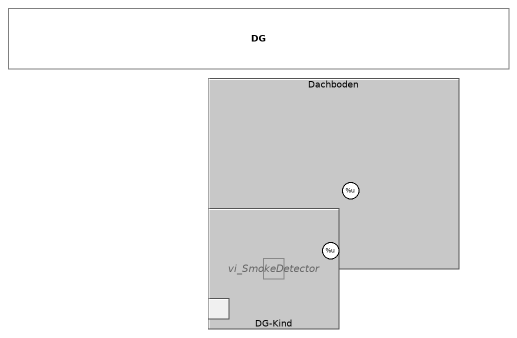
rectangle at (130,0)-(631,61): text "DG"
button at (330,70)-(581,261): text "Dachboden"; opens vi_Dachboden
button at (330,200)-(461,321): text "DG-Kind"; opens vi_DgKind
embedded screen at (440,230)-(461,251): vi_Lamp_tiny
embedded screen at (460,170)-(481,191): vi_Lamp_tiny
embedded screen at (385,250)-(406,271): vi_SmokeDetector
embedded screen at (330,290)-(351,311): vi_ButtonSingle_tiny
*)

(* Visualisation VI_EG
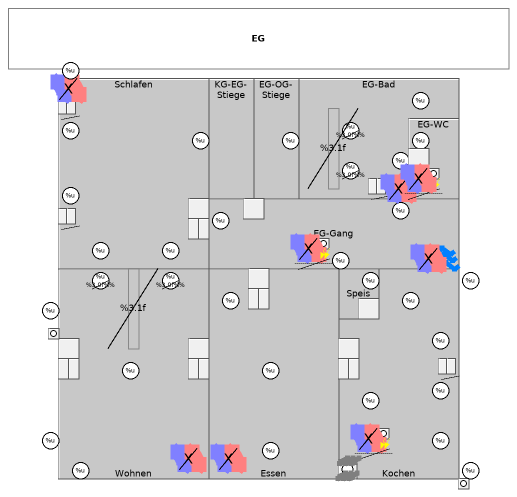
rectangle at (130,0)-(631,61): text "EG"
button at (460,260)-(581,471): text "Kochen"; opens vi_Kochen
button at (460,260)-(501,311): text "Speis"; opens vi_Speis
button at (330,260)-(461,471): text "Essen"; opens vi_Essen
button at (330,190)-(581,261): text "EG-Gang"; opens vi_EgGang
button at (420,70)-(581,191): text "EG-Bad"; opens vi_EgBad
button at (375,70)-(421,191): text "EG-OG- / Stiege"; opens vi_EgOgStiege
button at (530,110)-(581,191): text "EG-WC"; opens vi_EgWC
button at (330,70)-(376,191): text "KG-EG- / Stiege"; opens vi_KgEgStiege
button at (180,260)-(331,471): text "Wohnen"; opens vi_Wohnen
button at (180,70)-(331,261): text "Schlafen"; opens vi_Schlafen
embedded screen at (365,190)-(386,211): vi_ButtonSingle_tiny
embedded screen at (280,230)-(301,251): vi_Lamp_tiny
embedded screen at (210,230)-(231,251): vi_Lamp_tiny
embedded screen at (180,175)-(201,196): vi_Lamp_tiny
embedded screen at (180,110)-(201,131): vi_Lamp_tiny
embedded screen at (310,120)-(331,141): vi_Lamp_tiny
embedded screen at (310,190)-(331,231): vi_ButtonTripple_tiny
embedded screen at (180,200)-(201,221): vi_ButtonDouble_tiny
embedded screen at (180,90)-(201,111): vi_ButtonDouble_tiny
embedded screen at (440,230)-(451,241): vi_Motion
embedded screen at (210,260)-(231,281): vi_LampDimmer_tiny
embedded screen at (240,350)-(261,371): vi_Lamp_tiny
embedded screen at (380,350)-(401,371): vi_Lamp_tiny
embedded screen at (380,430)-(401,451): vi_Lamp_tiny
embedded screen at (480,380)-(501,401): vi_Lamp_tiny
embedded screen at (550,420)-(571,441): vi_Lamp_tiny
embedded screen at (520,280)-(541,301): vi_Lamp_tiny
embedded screen at (480,260)-(501,281): vi_Lamp_tiny
embedded screen at (190,450)-(211,471): vi_Lamp_tiny
embedded screen at (510,190)-(531,211): vi_Lamp_tiny
embedded screen at (450,240)-(471,261): vi_Lamp_tiny
embedded screen at (330,200)-(351,221): vi_Lamp_tiny
embedded screen at (530,80)-(551,101): vi_Lamp_tiny
embedded screen at (510,140)-(531,161): vi_Lamp_tiny
embedded screen at (530,120)-(551,141): vi_Lamp_tiny
embedded screen at (370,260)-(391,301): vi_ButtonTripple_tiny
embedded screen at (310,330)-(331,371): vi_ButtonTripple_tiny
embedded screen at (180,330)-(201,371): vi_ButtonTripple_tiny
embedded screen at (460,330)-(481,371): vi_ButtonTripple_tiny
embedded screen at (560,350)-(581,371): vi_ButtonDouble_tiny
embedded screen at (490,170)-(511,191): vi_ButtonDouble_tiny
embedded screen at (530,140)-(551,161): vi_ButtonSingle_tiny
embedded screen at (550,160)-(561,171): vi_Motion
embedded screen at (340,280)-(361,301): vi_Lamp_tiny
embedded screen at (180,70)-(201,91): vi_Temperature
embedded screen at (300,440)-(321,461): vi_Temperature
embedded screen at (340,440)-(361,461): vi_Temperature
embedded screen at (510,170)-(531,191): vi_Temperature
embedded screen at (420,230)-(441,251): vi_Temperature
embedded screen at (420,240)-(451,261): vi_Light
embedded screen at (500,420)-(511,431): vi_Motion
embedded screen at (480,420)-(501,441): vi_Temperature
embedded screen at (480,430)-(511,451): vi_Light
embedded screen at (530,170)-(561,191): vi_Light
embedded screen at (530,160)-(551,181): vi_Temperature
embedded screen at (580,470)-(591,481): vi_Motion
embedded screen at (170,320)-(181,331): vi_Motion
embedded screen at (580,260)-(601,281): vi_Lamp_tiny
embedded screen at (580,450)-(601,471): vi_Lamp_tiny
embedded screen at (160,420)-(181,441): vi_Lamp_tiny
embedded screen at (160,290)-(181,311): vi_Lamp_tiny
embedded screen at (180,50)-(201,71): vi_Lamp_tiny
embedded screen at (400,120)-(421,141): vi_Lamp_tiny
embedded screen at (560,240)-(581,261): vi_Hygrometer
embedded screen at (540,240)-(561,261): vi_Temperature
embedded screen at (460,450)-(481,471): vi_Smoke
embedded screen at (550,370)-(571,391): vi_Lamp_tiny
embedded screen at (550,320)-(571,341): vi_Lamp_tiny
embedded screen at (480,290)-(501,311): vi_ButtonSingle_tiny
embedded screen at (280,260)-(301,281): vi_LampDimmer_tiny
curve at (230,260)-(280,340): text "%3.1f"; shows MAIN._dimmerWohnenN_intensity
embedded screen at (460,150)-(481,171): vi_LampDimmer_tiny
embedded screen at (460,110)-(481,131): vi_LampDimmer_tiny
curve at (430,100)-(480,180): text "%3.1f"; shows MAIN._dimmerEgBadSM_intensity
2 more shapes without text or variables
*)

(* Visualisation VI_EG_JALOUSIEN
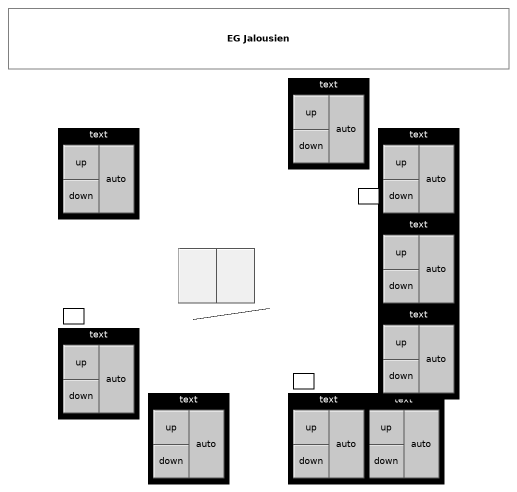
embedded screen at (300,240)-(391,311): vi_ButtonDouble_tiny
embedded screen at (180,120)-(261,211): VI_Jalousie_tiny
embedded screen at (180,320)-(261,411): VI_Jalousie_tiny
embedded screen at (270,385)-(351,476): VI_Jalousie_tiny
embedded screen at (485,385)-(566,476): VI_Jalousie_tiny
embedded screen at (410,385)-(491,476): VI_Jalousie_tiny
embedded screen at (500,300)-(581,391): VI_Jalousie_tiny
embedded screen at (500,210)-(581,301): VI_Jalousie_tiny
embedded screen at (500,120)-(581,211): VI_Jalousie_tiny
embedded screen at (410,70)-(491,161): VI_Jalousie_tiny
rectangle at (130,0)-(631,61): text "EG Jalousien"
3 more shapes without text or variables
*)

(* Visualisation EG/VI_EGGANG
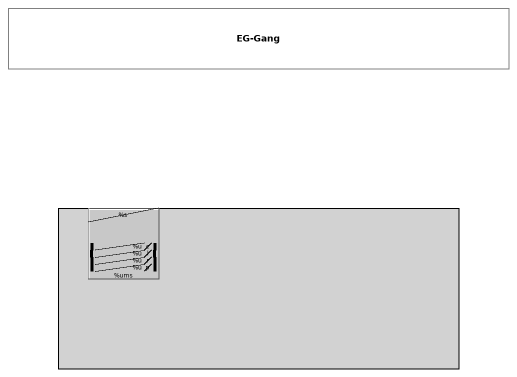
rectangle at (130,0)-(631,61): text "EG-Gang"
embedded screen at (210,200)-(281,271): vi_ButtonSingle
1 more shapes without text or variables
*)

(* Visualisation VI_GRAPH
1 elements of other kinds (tables, trends, ...) not read
*)

(* Visualisation KG/VI_HEIZEN
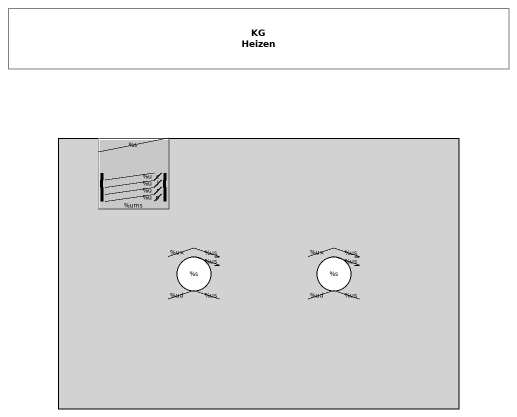
rectangle at (130,0)-(631,61): text "KG / Heizen"
embedded screen at (430,240)-(481,291): vi_Lamp
embedded screen at (290,240)-(341,291): vi_Lamp; dynamic style MAIN.viHeizenLicht
embedded screen at (220,130)-(291,201): vi_ButtonSingle
1 more shapes without text or variables
*)

(* Visualisation KG/VI_HOBBY
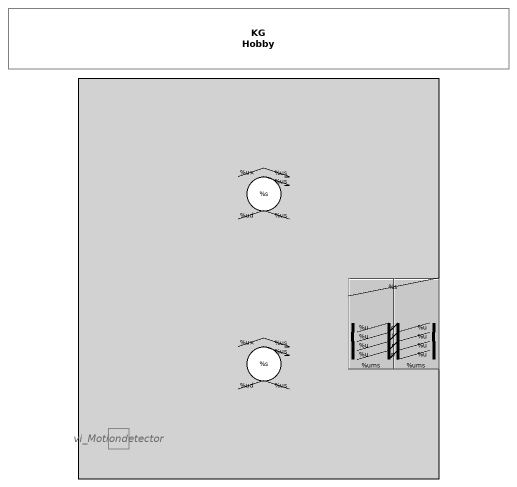
rectangle at (130,0)-(631,61): text "KG / Hobby"
embedded screen at (360,330)-(411,381): vi_Lamp
embedded screen at (360,160)-(411,211): vi_Lamp
embedded screen at (470,270)-(561,361): vi_ButtonDouble
embedded screen at (230,420)-(251,441): vi_Motiondetector
1 more shapes without text or variables
*)

(* Visualisation templates/vi_Hygrometer
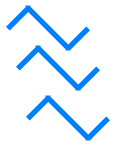
3 more shapes without text or variables
1 elements of other kinds (tables, trends, ...) not read
*)

(* Visualisation templates/VI_Jalousie_tiny
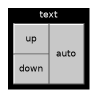
rectangle at (0,0)-(81,81): shows $FB_Jalousie$.viText
rectangle at (0,0)-(81,81): text "text"; shows $FB_Jalousie$.viText
button at (40,15)-(76,76): text "auto"; taps $FB_Jalousie$.viAuto
button at (5,45)-(41,76): text "down"; taps $FB_Jalousie$.viDown
button at (5,15)-(41,46): text "up"; taps $FB_Jalousie$.viUp
*)

(* Visualisation VI_KG
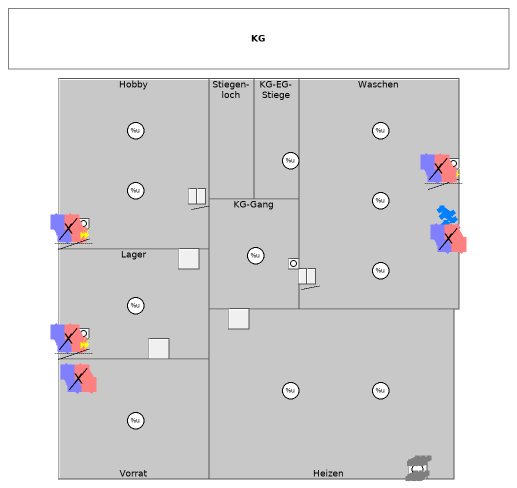
rectangle at (130,0)-(631,61): text "KG"
button at (325,300)-(576,471): text "Heizen"; opens vi_Heizen
button at (420,70)-(581,301): text "Waschen"; opens vi_Waschen
button at (330,190)-(421,301): text "KG-Gang"; opens vi_KgGang
button at (375,70)-(421,191): text "KG-EG- / Stiege"; opens vi_KgEgStiege
embedded screen at (365,235)-(386,256): vi_Lamp_tiny
embedded screen at (490,250)-(511,271): vi_Lamp_tiny
embedded screen at (490,180)-(511,201): vi_Lamp_tiny
embedded screen at (490,110)-(511,131): vi_Lamp_tiny
embedded screen at (400,140)-(421,161): vi_Lamp_tiny
embedded screen at (400,370)-(421,391): vi_Lamp_tiny
embedded screen at (490,370)-(511,391): vi_Lamp_tiny
embedded screen at (350,300)-(371,321): vi_ButtonSingle_tiny
embedded screen at (420,260)-(441,281): vi_ButtonDouble_tiny
embedded screen at (410,250)-(421,261): vi_Motion
button at (330,70)-(376,191): text "Stiegen- / loch"
button at (180,350)-(331,471): text "Vorrat"; opens vi_Vorrat
button at (180,240)-(331,351): text "Lager"; opens vi_Lager
button at (180,70)-(331,241): text "Hobby"; opens vi_Hobby
embedded screen at (245,400)-(266,421): vi_Lamp_tiny
embedded screen at (245,285)-(266,306): vi_Lamp_tiny
embedded screen at (245,170)-(266,191): vi_Lamp_tiny
embedded screen at (245,110)-(266,131): vi_Lamp_tiny
embedded screen at (270,330)-(291,351): vi_ButtonSingle_tiny
embedded screen at (300,240)-(321,261): vi_ButtonSingle_tiny
embedded screen at (310,180)-(331,201): vi_ButtonDouble_tiny
embedded screen at (200,210)-(211,221): vi_Motion
embedded screen at (200,320)-(211,331): vi_Motion
embedded screen at (570,150)-(581,161): vi_Motion
embedded screen at (550,160)-(581,181): vi_Light
embedded screen at (190,360)-(211,381): vi_Temperature
embedded screen at (180,210)-(201,231): vi_Temperature
embedded screen at (180,220)-(211,241): vi_Light
embedded screen at (180,320)-(201,341): vi_Temperature
embedded screen at (180,330)-(211,351): vi_Light
embedded screen at (530,450)-(551,471): vi_Smoke
embedded screen at (560,200)-(581,221): vi_Hygrometer
embedded screen at (560,220)-(581,241): vi_Temperature
embedded screen at (550,150)-(571,171): vi_Temperature
*)

(* Visualisation KG/VI_LAGER
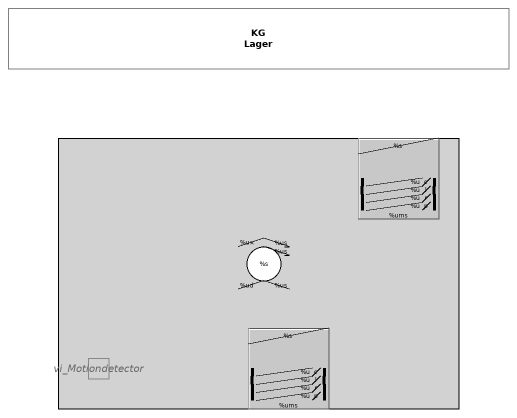
rectangle at (130,0)-(631,61): text "KG / Lager"
embedded screen at (480,130)-(561,211): vi_ButtonSingle
embedded screen at (360,230)-(411,281): vi_Lamp
embedded screen at (370,320)-(451,401): vi_ButtonSingle
embedded screen at (210,350)-(231,371): vi_Motiondetector
1 more shapes without text or variables
*)

(* Visualisation templates/VI_LAMP
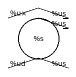
ellipse at (10,10)-(51,51): invisible if NOT $FB_Lamp$.FORCE
ellipse at (10,10)-(51,51): text "%s"; shows $FB_Lamp$.viText; alarm colour if $FB_Lamp$.Q; taps $FB_Lamp$.ON_OFF
curve at (30,50)-(60,60): text "%us"; shows $FB_Lamp$.usageTime / 1000
curve at (0,50)-(30,60): text "%ud"; shows $FB_Lamp$.usageDays
curve at (0,0)-(30,10): text "%u×"; shows $FB_Lamp$.usageCounterSwitchOn
curve at (30,0)-(60,10): text "%us"; shows $FB_Lamp$.viOnTimer / 1000
curve at (30,10)-(60,20): text "%us"; shows $FB_Lamp$.viOffTimer / 1000
curve at (55,10)-(60,10): invisible if NOT $FB_Lamp$.onTimer.Q
curve at (55,20)-(60,20): invisible if NOT $FB_Lamp$.offTimer.Q
*)

(* Visualisation templates/vi_Lamp_tiny
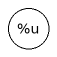
ellipse at (10,10)-(51,51): invisible if NOT $FB_Lamp$.FORCE
ellipse at (10,10)-(51,51): text "%u"; shows $FB_Lamp$.viOnTimer / 1000; alarm colour if $FB_Lamp$.Q; taps $FB_Lamp$.viOnOff
*)

(* Visualisation templates/vi_LampDimmer_tiny
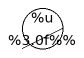
ellipse at (10,10)-(51,51): invisible if NOT $FB_Lamp$.FORCE
ellipse at (10,10)-(51,51): text "%u"; shows $FB_Lamp$.viOnTimer / 1000; alarm colour if $FB_Lamp$.Q; taps $FB_Lamp$.viOnOff
curve at (10,30)-(50,50): text "%3.0f%%"; shows $FB_Dimmer$.mIntensity
*)

(* Visualisation templates/vi_Light
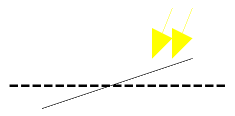
polyline at (0,50)-(150,100): text "-------------------"; invisible if NOT $FB_Light$.Error
2 more shapes without text or variables
1 elements of other kinds (tables, trends, ...) not read
*)

(* Visualisation templates/vi_Motion
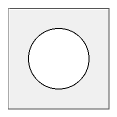
button at (0,0)-(101,101): taps $fbMotiondetector$.viIN
ellipse at (20,20)-(81,81): alarm colour if $fbMotiondetector$.myIN; taps $fbMotiondetector$.viIN
*)

(* Visualisation VI_OG
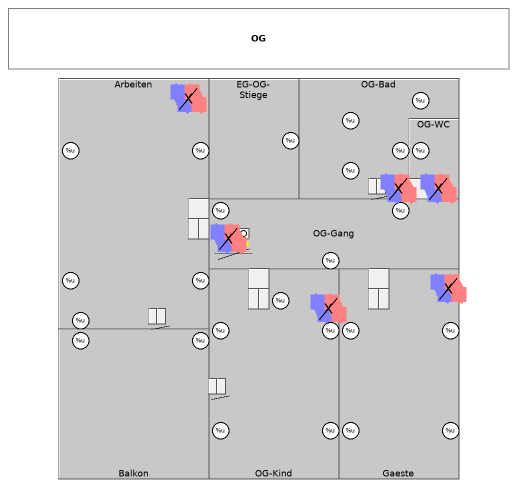
rectangle at (130,0)-(631,61): text "OG"
button at (460,260)-(581,471): text "Gaeste"; opens vi_Gaeste
button at (330,260)-(461,471): text "OG-Kind"; opens vi_OgKind
button at (330,190)-(581,261): text "OG-Gang"; opens vi_OgGang
button at (420,70)-(581,191): text "OG-Bad"; opens vi_OgBad
button at (330,70)-(421,191): text "EG-OG- / Stiege"; opens vi_EgOgStiege
button at (180,320)-(331,471): text "Balkon"; opens vi_Balkon
button at (180,70)-(331,321): text "Arbeiten"; opens vi_Arbeiten
button at (530,110)-(581,191): text "OG-WC"; opens vi_OgWC
embedded screen at (510,190)-(531,211): vi_Lamp_tiny
embedded screen at (440,240)-(461,261): vi_Lamp_tiny
embedded screen at (330,190)-(351,211): vi_Lamp_tiny
embedded screen at (360,220)-(371,231): vi_Motion
embedded screen at (490,260)-(511,301): vi_ButtonTripple_tiny
embedded screen at (460,310)-(481,331): vi_Lamp_tiny
embedded screen at (460,410)-(481,431): vi_Lamp_tiny
embedded screen at (560,310)-(581,331): vi_Lamp_tiny
embedded screen at (560,410)-(581,431): vi_Lamp_tiny
embedded screen at (330,370)-(351,391): vi_ButtonDouble_tiny
embedded screen at (270,300)-(291,321): vi_ButtonDouble_tiny
embedded screen at (370,260)-(391,301): vi_ButtonTripple_tiny
embedded screen at (310,190)-(331,231): vi_ButtonTripple_tiny
embedded screen at (490,170)-(511,191): vi_ButtonDouble_tiny
embedded screen at (530,170)-(551,191): vi_ButtonSingle_tiny
embedded screen at (560,270)-(581,291): vi_Temperature
embedded screen at (340,230)-(371,251): vi_Light
embedded screen at (440,290)-(461,311): vi_Temperature
embedded screen at (340,220)-(361,241): vi_Temperature
embedded screen at (550,170)-(571,191): vi_Temperature
embedded screen at (510,170)-(531,191): vi_Temperature
embedded screen at (530,130)-(551,151): vi_Lamp_tiny
embedded screen at (510,130)-(531,151): vi_Lamp_tiny
embedded screen at (460,150)-(481,171): vi_Lamp_tiny
embedded screen at (460,100)-(481,121): vi_Lamp_tiny
embedded screen at (530,80)-(551,101): vi_Lamp_tiny
embedded screen at (400,120)-(421,141): vi_Lamp_tiny
embedded screen at (310,130)-(331,151): vi_Lamp_tiny
embedded screen at (310,260)-(331,281): vi_Lamp_tiny
embedded screen at (180,260)-(201,281): vi_Lamp_tiny
embedded screen at (180,130)-(201,151): vi_Lamp_tiny
embedded screen at (310,320)-(331,341): vi_Lamp_tiny
embedded screen at (390,280)-(411,301): vi_Lamp_tiny
embedded screen at (330,410)-(351,431): vi_Lamp_tiny
embedded screen at (440,410)-(461,431): vi_Lamp_tiny
embedded screen at (440,310)-(461,331): vi_Lamp_tiny
embedded screen at (330,310)-(351,331): vi_Lamp_tiny
embedded screen at (300,80)-(321,101): vi_Temperature
embedded screen at (190,320)-(211,341): vi_Lamp_tiny
embedded screen at (190,300)-(211,321): vi_Lamp_tiny
*)

(* Visualisation VI_OG_JALOUSIEN
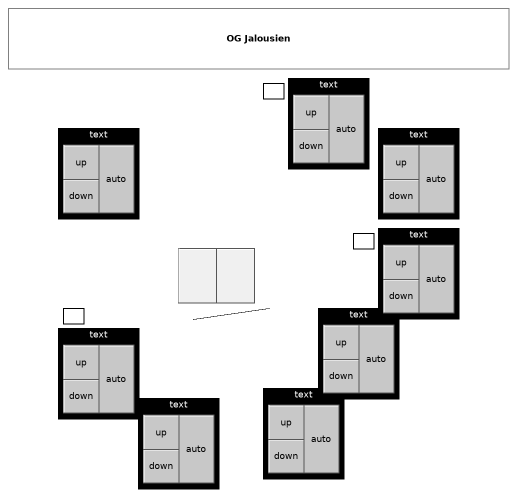
embedded screen at (300,240)-(391,311): vi_ButtonDouble_tiny
embedded screen at (180,120)-(261,211): VI_Jalousie_tiny
embedded screen at (180,320)-(261,411): VI_Jalousie_tiny
embedded screen at (260,390)-(341,481): VI_Jalousie_tiny
embedded screen at (385,380)-(466,471): VI_Jalousie_tiny
embedded screen at (440,300)-(521,391): VI_Jalousie_tiny
embedded screen at (500,220)-(581,311): VI_Jalousie_tiny
embedded screen at (500,120)-(581,211): VI_Jalousie_tiny
embedded screen at (410,70)-(491,161): VI_Jalousie_tiny
rectangle at (130,0)-(631,61): text "OG Jalousien"
3 more shapes without text or variables
*)

(* Visualisation OG/VI_OGGANG
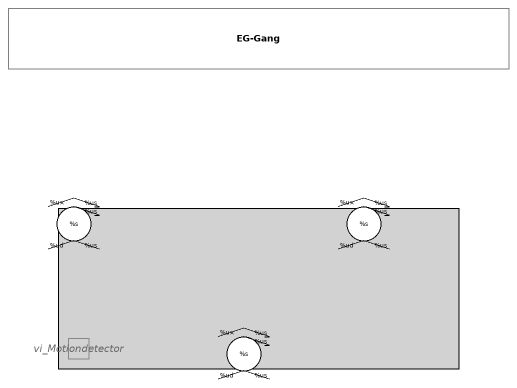
rectangle at (130,0)-(631,61): text "EG-Gang"
embedded screen at (190,330)-(211,351): vi_Motiondetector
embedded screen at (170,190)-(221,241): vi_Lamp; dynamic style MAIN.viHeizenLicht
embedded screen at (340,320)-(391,371): vi_Lamp; dynamic style MAIN.viHeizenLicht
embedded screen at (460,190)-(511,241): vi_Lamp; dynamic style MAIN.viHeizenLicht
1 more shapes without text or variables
*)

(* Visualisation EG/VI_SCHLAFEN
